Yaskawa INFORM job: FRONT_SEARCH_90ST-2_5040.JBI

/JOB
//NAME FRONT_SEARCH_90ST-2_5040
///FOLDERNAME 02-SKRZYNIE_JOBS
//POS
///NPOS 31,31,0,5,0,0
///TOOL 0
///POSTYPE PULSE
///PULSE
C00000=-24267,-14312,28258,73734,-14690,6801
C00001=-41484,-6818,29427,5360,-3449,36659
C00002=-41484,-6818,29427,5360,-3449,36659
///LIMIT ON
C00003=-41039,-6163,30067,9986,-3433,34548
///LIMIT OFF
C00004=-41484,-6818,29427,5360,-3449,36659
///LIMIT ON
C00005=-41484,-5631,32430,3998,-4621,37301
///LIMIT OFF
C00006=-41484,-6818,29427,5360,-3449,36659
C00007=-38039,-14917,11384,-18270,7506,47311
C00008=-20226,-24552,470,145490,-9534,-23074
C00009=-20665,-21162,6041,142737,-8292,-21815
C00010=-19901,-19164,7550,141930,-8950,-21348
C00011=-19516,-19775,3776,150210,-12864,-25491
C00012=-20078,-18914,166,160669,-19653,-31320
C00013=-20544,-20857,6268,142600,-8398,-21738
C00014=19451,-23723,-4446,126880,-27266,-2952
C00015=19498,-23692,-4078,126522,-27139,-2758
C00016=19135,-22655,-3320,127123,-27127,-3111
C00017=19251,-22842,-3139,126667,-27009,-2858
C00018=19251,-21966,-656,125111,-26336,-2039
C00019=19690,-24221,-4457,126204,-27147,-2571
C00020=19623,-34877,-16768,124729,-29078,51940
C00021=15304,-25293,-919,164625,-9673,28990
C00022=15060,-24487,-364,165662,-9870,28471
C00023=14820,-23667,211,166639,-10065,27982
C00024=14946,-24106,-99,166125,-9960,28239
C00025=14946,-23268,2164,165268,-9043,28646
C00026=15172,-24866,-626,165185,-9778,28711
C00027=22935,-43287,-23487,146875,-13252,38235
C00028=53252,-41973,-2905,102185,-37459,42403
C00029=0,-35574,42087,36666,-9339,1809
C00030=0,-52278,40443,0,6873,1
BC00000=922806
BC00001=954691
BC00002=954691
BC00003=954691
BC00004=954691
BC00005=954691
BC00006=954691
BC00007=954691
BC00008=954691
BC00009=954691
BC00010=954691
BC00011=954691
BC00012=954691
BC00013=954691
BC00014=954691
BC00015=954691
BC00016=954691
BC00017=954691
BC00018=954691
BC00019=954691
BC00020=954691
BC00021=954691
BC00022=954691
BC00023=954691
BC00024=954691
BC00025=954691
BC00026=954691
BC00027=941325
BC00028=895987
BC00029=781636
BC00030=774759
///POSTYPE BASE
///RECTAN
///RCONF 1,0,0,0,0,0,0,0,0,0,0,0,0,0,0,0,0,0,0,0,0,0,0,0
P00006=0.000,0.000,0.000,0.0000,0.0000,0.0000
///RCONF 0,0,0,0,0,0,0,0,0,0,0,0,0,0,0,0,0,0,0,0,0,0,0,0
P00501=-2.026,0.009,3.534,0.0000,0.0000,0.0000
///RCONF 1,0,0,0,0,0,0,0,0,0,0,0,0,0,0,0,0,0,0,0,0,0,0,0
P00502=-2.023,0.001,1.732,0.0000,0.0000,0.0000
P00503=0.138,-0.044,1.539,0.0000,0.0000,0.0000
P00504=-0.309,-0.010,1.636,0.0000,0.0000,0.0000
//INST
///DATE 2024/05/15 11:49
///ATTR SC,RW
///GROUP1 RB1,BS1
NOP
MOVJ C00000 BC00000 VJ=80.00
'::::::::::::::::::::::::::::::::
'W56 P
'::::::::::::::::::::::::::::::::
MOVL C00001 BC00001 V=500.0
MOVL C00002 BC00002 V=100.0 PL=0
REFP 3 C00003 BC00003
CALL JOB:SEARCH-R1
SET P0501 P0006
SFTON P0501
MOVL C00004 BC00004 V=166.7 PL=0
REFP 3 C00005 BC00005
CALL JOB:SEARCH-R1
SET P0501 P0006
SFTON P0501
MOVL C00006 BC00006 V=250.0 PL=0
MOVJ C00007 BC00007 VJ=10.00
SFTOF
'::::::::::::::::::::::::::::::::
'W56 L
'::::::::::::::::::::::::::::::::
MOVL C00008 BC00008 V=333.3
MOVL C00009 BC00009 V=100.0 PL=0
REFP 3 C00010 BC00010
CALL JOB:SEARCH-R1
SET P0502 P0006
SFTON P0502
MOVL C00011 BC00011 V=166.7 PL=0
REFP 3 C00012 BC00012
CALL JOB:SEARCH-R1
SET P0502 P0006
SFTON P0502
MOVL C00013 BC00013 V=250.0 PL=0
SFTOF
'::::::::::::::::::::::::::::::::
'W57 P
'::::::::::::::::::::::::::::::::
MOVL C00014 BC00014 V=500.0
MOVL C00015 BC00015 V=100.0 PL=0
REFP 3 C00016 BC00016
CALL JOB:SEARCH-R1
SET P0503 P0006
SFTON P0503
MOVL C00017 BC00017 V=166.7 PL=0
REFP 3 C00018 BC00018
CALL JOB:SEARCH-R1
SET P0503 P0006
SFTON P0503
MOVL C00019 BC00019 V=250.0 PL=0
SFTOF
'::::::::::::::::::::::::::::::::
'W57 L
'::::::::::::::::::::::::::::::::
MOVL C00020 BC00020 V=333.3
MOVL C00021 BC00021 V=500.0
MOVL C00022 BC00022 V=166.7 PL=0
REFP 3 C00023 BC00023
CALL JOB:SEARCH-R1
SET P0504 P0006
SFTON P0504
MOVL C00024 BC00024 V=166.7 PL=0
REFP 3 C00025 BC00025
CALL JOB:SEARCH-R1
SET P0504 P0006
SFTON P0504
MOVL C00026 BC00026 V=250.0 PL=0
SFTOF
MOVJ C00027 BC00027 VJ=50.00
MOVJ C00028 BC00028 VJ=50.00
MOVJ C00029 BC00029 VJ=80.00
MOVJ C00030 BC00030 VJ=80.00
END
